// TIA Portal project "home" (V15)

(* hardware
DEVICE "S7300/ET200M station_1"  S7-300 station
   slot 0: "Rail_0"  Rail  6ES7 390-1***0-0AA0
   slot 2: "PLC_1"  CPU 315-2 PN/DP  6ES7 315-2EH14-0AB0  V3.2
      slot 2: "PROFINET interface_1"  PN-IO
         slot 1: "Port_1"  Port
         slot 2: "Port_2"  Port
   slot 4: "DI 16/DO 16x24VDC/0.5A_1"  DI16/DO16 x 24V / 0.5A  6ES7 323-1BL00-0AA0
*)

// ===== PLC "PLC_1"  CPU 315-2 PN/DP =====

VAR_GLOBAL   // PLC tag table "Default tag table"
   "Tag_1" AT %MW200 : Int;
   "Tag_2" AT %M100.0 : Bool;
   "Tag_3" AT %MW10 : Int;
   "Tag_4" AT %Q0.0 : Bool;
   "Tag_5" AT %M0.0 : Bool;
   "Tag_6" AT %M0.1 : Bool;
END_VAR

DATA_BLOCK "WEB_DATA"   // DB1
{ S7_Optimized_Access := 'FALSE' }
VERSION : 0.1
   VAR
      "WORD" : Word;
      SZELEP1 : Bool;
      HETFO : Bool;
      KEDD : Bool;
      SZERDA : Bool;
      CSUTORTOK : Bool;
      PENTEK : Bool;
      SZOMBAT : Bool;
      VASARNAP : Bool;
      HETFO_FROM : String[10];
      KEDD_FROM : String[10];
      SZERDA_FROM : String[10];
      CSUTORTOK_FROM : String[10];
      PENTEK_FROM : String[10];
      SZOMBAT_FROM : String[10];
      VASARNAP_FROM : String[10];
      HETFO_TO : String[10];
      KEDD_TO : String[10];
      SZERDA_TO : String[10];
      CSUTORTOK_TO : String[10];
      PENTEK_TO : String[10];
      SZOMBAT_TO : String[10];
      VASARNAP_TO : String[10];
   END_VAR
BEGIN
END_DATA_BLOCK

// folder: SystemBlocksFolder/ReportSystemErrorFolder

DATA_BLOCK "RSE_DIAGNOSTIC_STATUS_DB"   // DB127
TITLE = Report System Error Diagnostic Block
{ S7_Optimized_Access := 'FALSE' }
AUTHOR : SIMATIC
FAMILY : RSEDIAG
NAME : RSE7
VERSION : 1.0
// This DB is part of report system error and will be updated by the RSE FB.
//  It is an interface for support of system diagnosis via the CPU web server.
   VAR
      Directory : Struct
         D_Version : Word := WORD#16#0100;   // Version that supports RSE
         D_pGlobalState : Word := WORD#16#0010;   // Byte offset to the start of the "GlobalState" section
         D_pQuery : Word := WORD#16#0014;   // Byte offset to the start of the "Query" section
         D_pComponent : Word := WORD#16#0020;   // Byte offset to the start of the "Component" section
         D_pError : Word := WORD#16#0024;   // Byte offset to the start of the "Error" section
         D_pState : Word := WORD#16#0028;   // Byte offset to the start of the "State" section
         D_pAlarm : Word := WORD#16#005A;   // Byte offset to the start of the "Alarm" section
         D_pSubComponent : Word := WORD#16#0082;   // Byte offset to the start of the "Subcomponent" section
      END_STRUCT;
      GlobalState : Struct
         G_EventCount : Word := WORD#16#0000;   // ID of the last event (counter)
         G_StartReporting : Bool := FALSE;   // Startup evaluation running
      END_STRUCT;
      Query : Struct
         Q_ClientID_User : DWord := DWORD#16#0000_0000;   // ID of the client
         Q_ClientID_Intern : DWord := DWORD#16#0000_0000;   // ID of the client (internal)
         Q_WithSubComponent : Bool := FALSE;   // With/without status of the underlying components (slower)
         Q_SubComponentAlarm : Bool := FALSE;   // AS-iMaster gibt AS-iSlave Alarme zurück
         Q_Reserved2 : Bool := FALSE;   // Reserved
         Q_Reserved3 : Bool := FALSE;   // Reserved
         Q_Reserved4 : Bool := FALSE;   // Reserved
         Q_Reserved5 : Bool := FALSE;   // Reserved
         Q_Reserved6 : Bool := FALSE;   // Reserved
         Q_Reserved7 : Bool := FALSE;   // Reserved
         Q_Start : Bool := FALSE;   // Start query
         Q_Error : Byte := BYTE#16#00;   // Internal error in query
         Q_Reserved8 : Byte := BYTE#16#00;   // Reserved
      END_STRUCT;
      Component : Struct
         C_AddressMode : Byte := BYTE#16#00;   // Addressing mode of the module
         C_Reserved1 : Byte := BYTE#16#00;   // Reserved
         C_ComponentID : Word := WORD#16#0000;   // Hardware ID of the component (internal)
      END_STRUCT;
      Error : Struct
         E_ErrorNo : Word := WORD#16#0000;   // Index of the requested/actual error
         E_LastError : Bool := FALSE;   // TRUE, if E_ErrorNo contains the indes of the last error, otherwise FALSE
      END_STRUCT;
      State : Struct
         S_Hierarchy : Byte := BYTE#16#00;   // Reserved
         S_Periphery : Byte := BYTE#16#00;   // Reserved
         S_SupFault : Bool := FALSE;   // The component is not obtainable
         S_NotAvailable : Bool := FALSE;   // The component does not exist
         S_Faulty : Bool := FALSE;   // The component is disrupted; the "Alarm" section is not empty
         S_MoreErrors : Bool := FALSE;   // There are more errors than RSE can store.
         S_Maintenance1 : Bool := FALSE;   // Maintenance required is indicated
         S_Maintenance2 : Bool := FALSE;   // Maintenance demand is indicated
         S_Deactivated : Bool := FALSE;   // The component was deactivated
         S_Reserved2 : Bool := FALSE;   // Reserved
         S_SubFault : Bool := FALSE;   // An underlying component is disrupted
         S_SubMaintenance1 : Bool := FALSE;   // Maintenance required is indicated for an underlying component
         S_SubMaintenance2 : Bool := FALSE;   // Maintenance demand is indicated for an underlying component
         S_SubDeactivated : Bool := FALSE;   // At least one lower-level component is disabled
         S_Reserved4 : Bool := FALSE;   // Reserved
         S_Reserved5 : Bool := FALSE;   // Reserved
         S_Reserved6 : Bool := FALSE;   // Reserved
         S_Reserved7 : Bool := FALSE;   // Reserved
         S_TIAMS : DWord := DWORD#16#0000_0000;   // Maintenance state of the component
         S_TIAMSChannelExist : DWord := DWORD#16#0000_0000;   // Maintenance state: Configured channels
         S_TIAMSChannelOK : DWord := DWORD#16#0000_0000;   // Maintenance State: Disrupted channels
         S_ChannelCount : Word := WORD#16#0000;   // Number of channels; Valid only when Q_WithSubComponent is set
         S_ChannelVector : Array[0..255] of Bool;   // List of channels involved; Valid only when Q_WithSubComponent is set
      END_STRUCT;
      Alarm : Struct
         A_ComponentID : Word := WORD#16#0000;   // Hardware ID of the component (internal)
         A_TextID1 : Word := WORD#16#0000;   // ID of the first error text
         A_TextLexikonID1 : Word := WORD#16#0000;   // ID of the first error text lexicon
         A_HelpTextLexikonID1 : Word := WORD#16#0000;   // ID of the first help text lexicon
         A_MapTextID : Word := WORD#16#0000;   // ID of the first error text in the export file (HMI)
         A_MapHelpTextID : Word := WORD#16#0000;   // ID of the first help text in the export file (HMI)
         A_TextID2 : Word := WORD#16#0000;   // ID of the second error text
         A_TextLexikonID2 : Word := WORD#16#0000;   // ID of the second error text lexicon
         A_HelpTextLexikonID2 : Word := WORD#16#0000;   // ID of the second help text lexicon
         A_MapTextID2 : Word := WORD#16#0000;   // ID of the second error text in the export file (HMI)
         A_MapHelpTextID2 : Word := WORD#16#0000;   // ID of the second help text in the export file (HMI)
         A_AlarmID : DWord := DWORD#16#0000_0000;   // Message number
         A_ValueCount : Word := WORD#16#000C;   // Number of other occupied bytes
         A_AssociatedValue : Array[1..6] of Word;   // Associated values of the message
      END_STRUCT;
      SubComponent : Struct
         U_SubComponentCount : Word := WORD#16#0000;   // Number of underlying components
         U_SubComponentFault : Array[1..4] of Byte;   // List of status of subordinate components, 1 byte per component
      END_STRUCT;
   END_VAR
BEGIN
END_DATA_BLOCK

// folder: (top level)

FUNCTION "Napok" : Void   // FC1, LAD
{ S7_Optimized_Access := 'FALSE' }
VERSION : 0.1
BEGIN

REGION Network 2 (STL)
         try   git;
END_REGION
END_FUNCTION

ORGANIZATION_BLOCK "Main"   // OB1, LAD
TITLE = "Main Program Sweep (Cycle)"
{ S7_Optimized_Access := 'FALSE' }
VERSION : 0.1
   VAR_TEMP
      OB1_EV_CLASS : Byte;   // Bits 0-3 = 1 (Coming event), Bits 4-7 = 1 (Event class 1)
      OB1_SCAN_1 : Byte;   // 1 (Cold restart scan 1 of OB 1), 3 (Scan 2-n of OB 1)
      OB1_PRIORITY : Byte;   // Priority of OB Execution
      OB1_OB_NUMBR : Byte;   // 1 (Organization block 1, OB1)
      OB1_RESERVED_1 : Byte;   // Reserved for system
      OB1_RESERVED_2 : Byte;   // Reserved for system
      OB1_PREV_CYCLE : Int;   // Cycle time of previous OB1 scan (milliseconds)
      OB1_MIN_CYCLE : Int;   // Minimum cycle time of OB1 (milliseconds)
      OB1_MAX_CYCLE : Int;   // Maximum cycle time of OB1 (milliseconds)
      OB1_DATE_TIME : Date_And_Time;   // Date and time OB1 started
   END_VAR
BEGIN

REGION Network 1
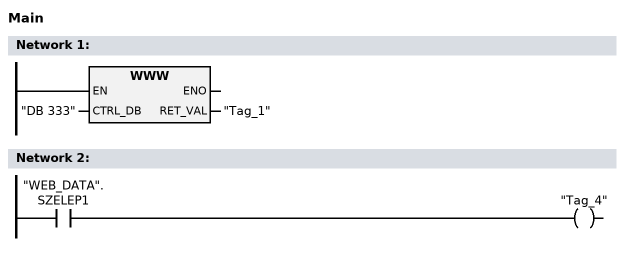
   "Tag_1" := WWW(CTRL_DB := "DB 333");
END_REGION

REGION Network 2
   RUNG wire#powerrail
      Contact( "WEB_DATA".SZELEP1 )
      Coil( "Tag_4" )
   END_RUNG
   // the same network as SCL:
   "Tag_4" := "WEB_DATA".SZELEP1;
END_REGION

REGION Network 3 (STL): Call system diagnostics block
         CALL  "RSE_FB", "RSE_DB";
END_REGION
END_ORGANIZATION_BLOCK

ORGANIZATION_BLOCK "I/O_FLT1"   // OB82, STL
TITLE = "I/O Point Fault"
{ S7_Optimized_Access := 'FALSE' }
VERSION : 0.1
   VAR_TEMP
      OB82_EV_CLASS : Byte;   // 16#39, Event class 3, Entering event state, Internal fault event
      OB82_FLT_ID : Byte;   // 16#XX, Fault identifcation code
      OB82_PRIORITY : Byte;   // Priority of OB Execution
      OB82_OB_NUMBR : Byte;   // 82 (Organization block 82, OB82)
      OB82_RESERVED_1 : Byte;   // Reserved for system
      OB82_IO_FLAG : Byte;   // Input (01010100), Output (01010101)
      OB82_MDL_ADDR : Word;   // Base address of module with fault
      OB82_MDL_DEFECT : Bool;   // Module defective
      OB82_INT_FAULT : Bool;   // Internal fault
      OB82_EXT_FAULT : Bool;   // External fault
      OB82_PNT_INFO : Bool;   // Point information
      OB82_EXT_VOLTAGE : Bool;   // External voltage low
      OB82_FLD_CONNCTR : Bool;   // Field wiring connector missing
      OB82_NO_CONFIG : Bool;   // Module has no configuration data
      OB82_CONFIG_ERR : Bool;   // Module has configuration error
      OB82_MDL_TYPE : Byte;   // Type of module
      OB82_SUB_MDL_ERR : Bool;   // Sub-Module is missing or has error
      OB82_COMM_FAULT : Bool;   // Communication fault
      OB82_MDL_STOP : Bool;   // Module is stopped
      OB82_WTCH_DOG_FLT : Bool;   // Watch dog timer stopped module
      OB82_INT_PS_FLT : Bool;   // Internal power supply fault
      OB82_PRIM_BATT_FLT : Bool;   // Primary battery is in fault
      OB82_BCKUP_BATT_FLT : Bool;   // Backup battery is in fault
      OB82_RESERVED_2 : Bool;   // Reserved for system
      OB82_RACK_FLT : Bool;   // Rack fault, only for bus interface module
      OB82_PROC_FLT : Bool;   // Processor fault
      OB82_EPROM_FLT : Bool;   // EPROM fault
      OB82_RAM_FLT : Bool;   // RAM fault
      OB82_ADU_FLT : Bool;   // ADU fault
      OB82_FUSE_FLT : Bool;   // Fuse fault
      OB82_HW_INTR_FLT : Bool;   // Hardware interupt input in fault
      OB82_RESERVED_3 : Bool;   // Reserved for system
      OB82_DATE_TIME : Date_And_Time;   // Date and time OB82 started
   END_VAR
BEGIN

REGION Network 1: Call system diagnostics block
         CALL  "RSE_FB", "RSE_DB";
END_REGION
END_ORGANIZATION_BLOCK

ORGANIZATION_BLOCK "I/O_FLT2"   // OB83, STL
TITLE = "I/O Point Fault"
{ S7_Optimized_Access := 'FALSE' }
VERSION : 0.1
   VAR_TEMP
      OB83_EV_CLASS : Byte;   // 16#38/39, Event class 3, module inserted/removed (8/9)
      OB83_FLT_ID : Byte;   // 16#XX, Fault identifcation code
      OB83_PRIORITY : Byte;   // Priority of OB Execution
      OB83_OB_NUMBR : Byte;   // 83 (Organization block 83, OB83)
      OB83_RESERVED_1 : Byte;   // Reserved for system
      OB83_MDL_ID : Byte;   // Input module (01010100), Output module (01010101)
      OB83_MDL_ADDR : Word;   // Base address of module with point fault
      OB83_RACK_NUM : Int;   // Number of rack that has module with point fault
      OB83_MDL_TYPE : Word;   // Module type with point fault
      OB83_DATE_TIME : Date_And_Time;   // Date and time OB83 started
   END_VAR
BEGIN

REGION Network 1: Call system diagnostics block
         CALL  "RSE_FB", "RSE_DB";
END_REGION
END_ORGANIZATION_BLOCK

ORGANIZATION_BLOCK "OBNL_FLT"   // OB85, STL
TITLE = "Organization Block (OB) Not Loaded Fault"
{ S7_Optimized_Access := 'FALSE' }
VERSION : 0.1
   VAR_TEMP
      OB85_EV_CLASS : Byte;   // 16#35 Event class 3
      OB85_FLT_ID : Byte;   // 16#XX, Fault identification code
      OB85_PRIORITY : Byte;   // Priority of OB Execution
      OB85_OB_NUMBR : Byte;   // 85 (Organization block 85, OB85)
      OB85_RESERVED_1 : Byte;   // Reserved for system
      OB85_RESERVED_2 : Byte;   // Reserved for system
      OB85_RESERVED_3 : Int;   // Reserved for system
      OB85_ERR_EV_CLASS : Byte;   // Class of event causing error
      OB85_ERR_EV_NUM : Byte;   // Number of event causing error
      OB85_OB_PRIOR : Byte;   // Priority of OB causing error
      OB85_OB_NUM : Byte;   // Number of OB causing error
      OB85_DATE_TIME : Date_And_Time;   // Date and time OB85 started
   END_VAR
BEGIN

REGION Network 1
         L     b#16#A1;  //
         L     #OB85_FLT_ID;
         ==I;
         JC    K_OB;
         L     b#16#A2;  //
         ==I;
         JC    K_OB;
         L     b#16#A3;  //
         L     #OB85_FLT_ID;
         ==I;
         JC    K_B;
         JU    F_PA;
END_REGION

REGION Network 2
   K_OB: JU    STOP;
         JU    ENDE;
END_REGION

REGION Network 3
   K_B:  JU    STOP;
         JU    ENDE;
END_REGION

REGION Network 4
   F_PA: NOP   0;
         JU    ENDE;
END_REGION

REGION Network 5
   STOP: CALL  STP;
END_REGION

REGION Network 6

   //

   ENDE: NOP   0;
END_REGION
END_ORGANIZATION_BLOCK

ORGANIZATION_BLOCK "RACK_FLT"   // OB86, STL
TITLE = "Loss Of Rack Fault"
{ S7_Optimized_Access := 'FALSE' }
VERSION : 0.1
   VAR_TEMP
      OB86_EV_CLASS : Byte;   // 16#38/39 Event class 3
      OB86_FLT_ID : Byte;   // 16#C1/C4/C5, Fault identification code
      OB86_PRIORITY : Byte;   // Priority of OB Execution
      OB86_OB_NUMBR : Byte;   // 86 (Organization block 86, OB86)
      OB86_RESERVED_1 : Byte;   // Reserved for system
      OB86_RESERVED_2 : Byte;   // Reserved for system
      OB86_MDL_ADDR : Word;   // Base address of IM module in rack with fault
      OB86_RACKS_FLTD : Array[0..31] of Bool;   // Racks in fault
      OB86_DATE_TIME : Date_And_Time;   // Date and time OB86 started
   END_VAR
BEGIN

REGION Network 1: Call system diagnostics block
         CALL  "RSE_FB", "RSE_DB";
END_REGION
END_ORGANIZATION_BLOCK